RoboDK station: Cooking Station.rdk

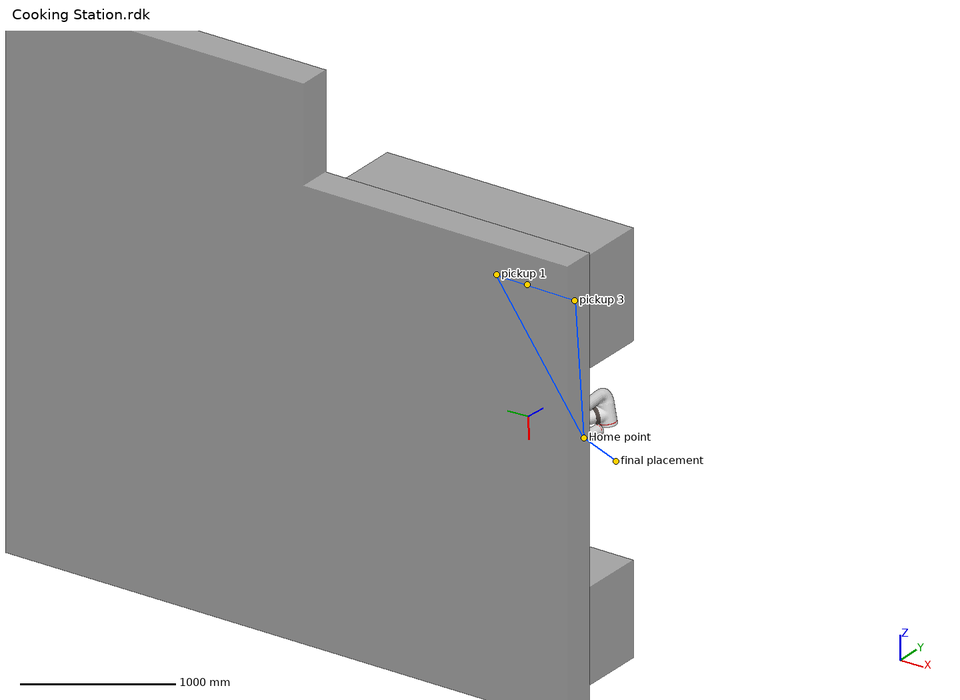
[picture v0: the station drawn from its stored meshes, robots at their saved joint values, targets as dots, program paths as lines]
Station Cooking Station (saved by RoboDK 5.8.0). Poses are relative to the parent item; angles as X-Y-Z fixed-axis rotations.
  - object Layout-1 (with pedestal) - cobot-pedestal-1 at (0, 0, 0) mm, size 200 x 850 x 200 mm, geometry from Layout-1 (with pedestal) - cobot-pedestal-1.STL
  - object Layout-1 (with pedestal) - fridge-1 at (0, 0, 0) mm, size 1550 x 842 x 700 mm, geometry from Layout-1 (with pedestal) - fridge-1.STL
  - object Layout-1 (with pedestal) - noodle-station-1 at (0, 0, 0) mm, size 1930 x 835 x 810 mm, geometry from Layout-1 (with pedestal) - noodle-station-1.STL
  - object Layout-1 (with pedestal) - robot-room-floorplan-1 at (0, 0, 0) mm, size 4410 x 250 x 4005 mm, geometry from Layout-1 (with pedestal) - robot-room-floorplan-1.STL
  - frame ERA5 Base at (3489.33, 905.22, 1594.26) mm, rotated rx -127.5 ry 87.08 rz -37.47 deg
    - robot ERA5 (model FAIRINO FR5): 6 axes
        modified DH rows (alpha deg, a mm, theta deg, d mm): 0, 0, 0, 152; 90, 0, 180, 0; 0, 425, 0, 0; 0, 395, 0, 130; -90, 0, 0, 102; 90, 0, 180, 100
        joint limits [-175, -265, -160, -265, -175, -175] to [175, 85, 160, 85, 175, 175]; home [0, -90, -90, 0, 90, 0]; saved at [79.951, -55.942, 136.29, -170.304, -90.421, 96.035]
    - target Home point (Cartesian target) at (56.41, -422.49, 14.62) mm, rotated rx -179.58 ry 0 rz 73.92 deg; joints [79.951, -55.942, 136.29, -170.304, -90.42, 96.029] of ERA5
    - target pickup 1 (Cartesian target) at (-857.08, 341.18, 150.31) mm, rotated rx 179.86 ry -0.4 rz -177.13 deg; joints [-29.819, -12.041, 10.746, -89.116, -89.9, -122.684] of ERA5
    - target pickup 2 (Cartesian target) at (-844.39, 100.09, 149.73) mm, rotated rx 179.86 ry -0.4 rz -177.13 deg; joints [-15.554, -31.411, 49.787, -108.799, -90.004, -108.42] of ERA5
    - target pickup 3 (Cartesian target) at (-822.87, -274.34, 148.81) mm, rotated rx 179.86 ry -0.4 rz -177.13 deg; joints [9.84, -28.283, 43.734, -105.832, -90.185, -83.026] of ERA5
    - target final placement (Cartesian target) at (139.24, -702.39, -23.28) mm, rotated rx -179.58 ry 0 rz 73.94 deg; joints [-68.28, -146.715, -84.537, -39.007, 89.668, 127.784] of ERA5
  - program Prog1 (8 instructions, listed below)
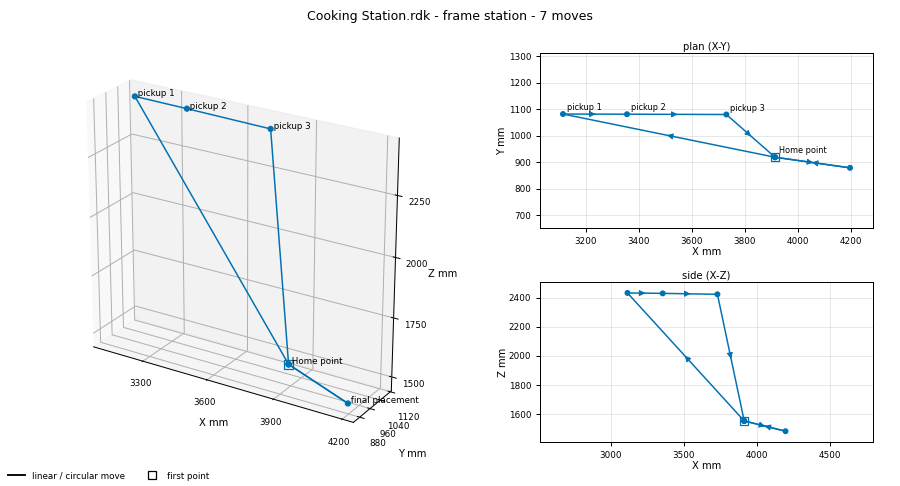
[picture p0: tool path of Cooking Station.rdk in frame station, 7 of 7 moves have a stored position in this frame; points joined in program order, loops and branches not executed]

--- program Prog1 (robot ERA5) ---
  Set Ref.: ERA5 Base
  MoveL (Home point)
  MoveL (pickup 1)
  MoveL (pickup 2)
  MoveL (pickup 3)
  MoveL (Home point)
  MoveL (final placement)
  MoveL (Home point)
